{attribute 'GeneratedUsingTerminal: EL4122--0000'}
{attribute addProperty BoxType "EL4122--0000"}
{attribute addProperty Id "Channel_1AT %Q*Channel_5F9B7EA62Channel_2AT %Q*Channel_5F9B7EA62WcStateAT %I*WcState_0B2B16F91InfoDataAT %I*InfoData_94A18F5E2"}
{attribute addProperty CRC "3722317115"}
{attribute addProperty Size "7"}
TYPE EL4122_DDDE0D3B EXTENDS EtcSlaveTerminalBase_947E5A46 :
STRUCT
	{attribute addProperty Name "Channel_1"}
	Channel_1 : Channel_5F9B7EA6;
	{attribute addProperty Name "Channel_2"}
	Channel_2 : Channel_5F9B7EA6;
	{attribute addProperty Name "WcState"}
	WcState : WcState_0B2B16F9;
	{attribute addProperty Name "InfoData"}
	InfoData : InfoData_94A18F5E;
END_STRUCT
END_TYPE

(* stored: Version 1.2.0.0, ProductVersion 3.1.4024.9
   DUT EL4122_DDDE0D3B: Id {7268a861-5326-43bd-ac07-919baba62a1e} *)
